// TwinCAT 3 PLC project Sample03
// Title: StateSample03
// Company: Beckhoff Automation
// ProjectVersion: 1.0.0.0
// ProgramVersion: 3.1.4022.3
// libraries:
//   Tc2_Standard, * (Beckhoff Automation GmbH)
//   Tc2_System, * (Beckhoff Automation GmbH)
//   Tc3_Module, * (Beckhoff Automation GmbH)
// project tree:
//   / ClassDiagram.TcCD (not stored), PlcTask.TcTTO
//   POUs/ FB_CoinEjectedState.TcPOU, FB_HasCoinState.TcPOU, FB_Machine.TcPOU, I_State.TcIO, I_StateMachine.TcIO, MAIN.TcPOU, FB_ProductEjectedState.TcPOU, FB_WaitingState.TcPOU
//   Version/ Global_Version.TcGVL
// real-time tasks:
//   TASK PlcTask: cycle T#10ms, priority 20, ADS port 350

CONFIGURATION Sample03
    RESOURCE PLC ON TwinCAT3
        TASK PlcTask(INTERVAL := T#10ms, PRIORITY := 20);
        PROGRAM MAIN WITH PlcTask : MAIN;
    END_RESOURCE
END_CONFIGURATION

// ---- Version/Global_Version.TcGVL
{attribute 'TcGenerated'}
// This function has been automatically generated from the project information.
VAR_GLOBAL CONSTANT
	{attribute 'const_non_replaced'}
	{attribute 'linkalways'}
	stLibVersion_StateSample03 : ST_LibVersion := (iMajor := 1, iMinor := 0, iBuild := 0, iRevision := 0, sVersion := '1.0.0.0');
END_VAR

// ---- POUs/I_State.TcIO
INTERFACE I_State

METHOD CustomerTakesCoin : BOOL
VAR_INPUT
END_VAR
END_METHOD

METHOD CustomerTakesProduct : BOOL
VAR_INPUT
END_VAR
END_METHOD

PROPERTY Description : STRING
GET
END_GET
END_PROPERTY

METHOD InsertCoin : BOOL
VAR_INPUT
END_VAR
END_METHOD

METHOD PressButton : BOOL
VAR_INPUT
END_VAR
END_METHOD

END_INTERFACE

// ---- POUs/I_StateMachine.TcIO
INTERFACE INTERNAL I_StateMachine

PROPERTY INTERNAL nProducts : UINT
GET
END_GET
END_PROPERTY

METHOD INTERNAL SetProducts : BOOL
VAR_INPUT
	newProducts : UINT;
END_VAR
END_METHOD

METHOD INTERNAL SetState : BOOL
VAR_INPUT
	newState : I_State;
END_VAR
END_METHOD

END_INTERFACE

// ---- POUs/MAIN.TcPOU
PROGRAM MAIN
VAR
	fbMachine			:	FB_Machine(3);
	sState				:	STRING;
	bButton				:	BOOL;
	bInsertCoin			:	BOOL;
	bTakeProduct		:	BOOL;
	bTakeCoin			:	BOOL;
END_VAR

fbMachine(	bButton	:= bButton,
			bInsertCoin := bInsertCoin,
			bTakeProduct := bTakeProduct,
			bTakeCoin := bTakeCoin);
sState := fbMachine.ipState.Description;

bButton := FALSE;
bInsertCoin := FALSE;
bTakeProduct := FALSE;
bTakeCoin := FALSE;

END_PROGRAM

// ---- POUs/FB_Machine.TcPOU
FUNCTION_BLOCK PUBLIC FB_Machine IMPLEMENTS I_StateMachine
VAR_INPUT
	bButton				: BOOL;
	bInsertCoin			: BOOL;
	bTakeProduct 		:	BOOL;
	bTakeCoin 			:	BOOL;	
END_VAR
VAR_OUTPUT
	ipState				:	I_State := fbWaitingState;	
		
END_VAR
VAR
	fbCoinEjectedState		:	FB_CoinEjectedState;
	fbHasCoinState				:	FB_HasCoinState;
	fbProductEjectedState	:	FB_ProductEjectedState;
	fbWaitingState				:	FB_WaitingState;
	
	_nProducts			:	UINT;
	
	rtrigButton				:	R_TRIG;
	rtrigInsertCoin			:	R_TRIG;
	rtrigTakeProduct		:	R_TRIG;
	rtrigTakeCoin			:	R_TRIG;
END_VAR

rtrigButton(CLK := bButton);
rtrigInsertCoin(CLK := bInsertCoin);
rtrigTakeProduct(CLK := bTakeProduct);
rtrigTakeCoin(CLK := bTakeCoin);

IF (rtrigButton.Q) THEN
	ipState.PressButton();
END_IF

IF (rtrigInsertCoin.Q) THEN
	ipState.InsertCoin();
END_IF

IF (rtrigTakeProduct.Q) THEN
	ipState.CustomerTakesProduct();
END_IF

IF (rtrigTakeCoin.Q) THEN
	ipState.CustomerTakesCoin();
END_IF

PROPERTY INTERNAL CoinEjectedState : I_State
GET
CoinEjectedState := THIS^.fbCoinEjectedState;
END_GET
END_PROPERTY

METHOD FB_init : BOOL
VAR_INPUT
	bInitRetains : BOOL; // if TRUE, the retain variables are initialized (warm start / cold start)
	bInCopyCode : BOOL;  // if TRUE, the instance afterwards gets moved into the copy code (online change)
	nProducts :	UINT;
END_VAR
THIS^._nProducts := nProducts;

wireUpStateTransitions();
END_METHOD

PROPERTY INTERNAL HasCoinState : I_State
GET
HasCoinState := THIS^.fbHasCoinState;
END_GET
END_PROPERTY

PROPERTY INTERNAL nProducts : UINT
GET
nProducts := _nProducts;
END_GET
END_PROPERTY

PROPERTY INTERNAL ProductEjectedState : I_State
GET
ProductEjectedState := THIS^.fbProductEjectedState;
END_GET
END_PROPERTY

METHOD INTERNAL SetProducts : BOOL
VAR_INPUT
	newProducts : UINT;
END_VAR
THIS^._nProducts := newProducts;
END_METHOD

METHOD INTERNAL SetState : BOOL
VAR_INPUT
	newState : I_State;
END_VAR
THIS^.ipState := newState;
END_METHOD

PROPERTY INTERNAL WaitingState : I_State
GET
WaitingState := THIS^.fbWaitingState;
END_GET
END_PROPERTY

METHOD PRIVATE wireUpStateTransitions
fbWaitingState.SetTransitionStates(
	Machine := THIS^,
	CoinInsertedNext := fbHasCoinState
);

fbHasCoinState.SetTransitionStates(
	Machine := THIS^,
	ButtonPressedProductDecrementedNext := fbProductEjectedState,
	ButtonPressedNoProductNext := fbCoinEjectedState
);

fbProductEjectedState.SetTransitionStates(
	Machine := THIS^,
	AfterProductEjectedNext := fbWaitingState
);

fbCoinEjectedState.SetTransitionStates(
	Machine := THIS^,
	CustomerTakesCoinNext := fbWaitingState
);
END_METHOD

END_FUNCTION_BLOCK

// ---- POUs/FB_CoinEjectedState.TcPOU
FUNCTION_BLOCK INTERNAL FB_CoinEjectedState IMPLEMENTS I_State
VAR_INPUT
END_VAR
VAR_OUTPUT
END_VAR
VAR
	pMachine : I_StateMachine;
	customerTakesCoinNext : I_State;
END_VAR

METHOD CustomerTakesCoin : BOOL
ADSLOGSTR(ADSLOG_MSGTYPE_HINT, 'Customer has taken the coin.', '');
pMachine.SetState( customerTakesCoinNext );
END_METHOD

METHOD CustomerTakesProduct : BOOL
END_METHOD

PROPERTY Description : STRING
GET
Description := 'Coin Ejected';
END_GET
END_PROPERTY

METHOD InsertCoin : BOOL
END_METHOD

METHOD PressButton : BOOL
END_METHOD

METHOD SetTransitionStates
VAR_INPUT
	Machine : I_StateMachine;
	CustomerTakesCoinNext : I_State;
END_VAR
THIS^.customerTakesCoinNext := CustomerTakesCoinNext;
THIS^.pMachine := Machine;
END_METHOD

END_FUNCTION_BLOCK

// ---- POUs/FB_HasCoinState.TcPOU
FUNCTION_BLOCK INTERNAL FB_HasCoinState IMPLEMENTS I_State
VAR_INPUT
END_VAR
VAR_OUTPUT
END_VAR
VAR
	pMachine : I_StateMachine;
	buttonPressedProductDecrementedNext : I_State;
	buttonPressedNoProductNext : I_State;
END_VAR

METHOD CustomerTakesCoin : BOOL
END_METHOD

METHOD CustomerTakesProduct : BOOL
END_METHOD

PROPERTY Description : STRING
GET
Description := 'Has Coin';
END_GET
END_PROPERTY

METHOD InsertCoin : BOOL
END_METHOD

METHOD PressButton : BOOL
IF (THIS^.pMachine.nProducts > 0) THEN
	THIS^.pMachine.SetProducts(THIS^.pMachine.nProducts - 1);
	ADSLOGSTR(ADSLOG_MSGTYPE_HINT, 'Customer has pressed the button. Output product.', '');
	pMachine.SetState(buttonPressedProductDecrementedNext);
ELSE				
	ADSLOGSTR(ADSLOG_MSGTYPE_HINT, 'Customer has pressed the button. No more products. Return coin.', '');
	pMachine.SetState(buttonPressedNoProductNext);
END_IF
END_METHOD

METHOD SetTransitionStates
VAR_INPUT
	Machine : I_StateMachine;
	ButtonPressedProductDecrementedNext : I_State;
	ButtonPressedNoProductNext : I_State;
END_VAR
THIS^.buttonPressedProductDecrementedNext := ButtonPressedProductDecrementedNext;
THIS^.buttonPressedNoProductNext := ButtonPressedNoProductNext;
THIS^.pMachine := Machine;
END_METHOD

END_FUNCTION_BLOCK

// ---- POUs/FB_ProductEjectedState.TcPOU
FUNCTION_BLOCK INTERNAL FB_ProductEjectedState IMPLEMENTS I_State
VAR_INPUT
END_VAR
VAR_OUTPUT
END_VAR
VAR
	pMachine : I_StateMachine;
	afterProductEjectedNext : I_State;
END_VAR

METHOD CustomerTakesCoin : BOOL
END_METHOD

METHOD CustomerTakesProduct : BOOL
ADSLOGSTR(ADSLOG_MSGTYPE_HINT, 'Customer has taken the product.', '');
pMachine.SetState(afterProductEjectedNext);
END_METHOD

PROPERTY Description : STRING
GET
Description := 'Product Ejected';
END_GET
END_PROPERTY

METHOD InsertCoin : BOOL
END_METHOD

METHOD PressButton : BOOL
END_METHOD

METHOD SetTransitionStates
VAR_INPUT
	Machine : I_StateMachine;
	AfterProductEjectedNext : I_State;
END_VAR
THIS^.afterProductEjectedNext := AfterProductEjectedNext;
THIS^.pMachine := Machine;
END_METHOD

END_FUNCTION_BLOCK

// ---- POUs/FB_WaitingState.TcPOU
FUNCTION_BLOCK INTERNAL FB_WaitingState IMPLEMENTS I_State
VAR_INPUT
END_VAR
VAR_OUTPUT
END_VAR
VAR
	pMachine : I_StateMachine;
	coinInsertedNext : I_State;
END_VAR

METHOD CustomerTakesCoin : BOOL
END_METHOD

METHOD CustomerTakesProduct : BOOL
END_METHOD

PROPERTY Description : STRING
GET
Description := 'Waiting';
END_GET
END_PROPERTY

METHOD InsertCoin : BOOL
ADSLOGSTR(ADSLOG_MSGTYPE_HINT, 'Customer has insert a coin.', '');
pMachine.SetState(coinInsertedNext);
END_METHOD

METHOD PressButton : BOOL
END_METHOD

METHOD SetTransitionStates
VAR_INPUT
	Machine : I_StateMachine;
	CoinInsertedNext : I_State;
END_VAR
THIS^.coinInsertedNext := CoinInsertedNext;
THIS^.pMachine := Machine;
END_METHOD

END_FUNCTION_BLOCK
